TYPE EOLFiberSwitchConfig EXTENDS DeviceConfiguration :
STRUCT
	SerialCommunication : SerialCommunication;
END_STRUCT
END_TYPE

(* stored: Version 1.1.0.1, ProductVersion 3.1.4024.4
   DUT EOLFiberSwitchConfig: Id {d9c2b2eb-46d7-4b62-9082-d3953504aece} *)
